Staubli VAL3: SettingGEN.dtx

num nCOLMAX = 39
num nCOLMIN
public num nColumn
public num nFocused
public num nListSize
num nROWMAX = 12
num nROWMIN
public num nRow
string sErrorMessage
string sErrorMsg[10]
  [1] = "An error has been detected in the Page library *\../*"
  [2] = "Variable sTxtBoxLen[*] has an illegal value"
  [3] = "Variable sTxtBoxPos[*] has an illegal value"
public string sFALSE = "FALSE"
public string sLabel[4]
  [0] = "-Calibrated pointer--"
  [1] = "-Event Logger --"
  [2] = "-Software --"
  [3] = "-Approach --"
public string sLabelPos[4]
  [0] = "0;0"
  [1] = "22;3"
  [2] = "22;0"
  [3] = "0;5"
public string sMenu = "; ; ; ENCODER DETECT CONVEYOR ; OK"
public string sTRUE = "TRUE"
public string sTitle
public string sTxtBoxAuthord[11]
  [0] = "0123456789.-"
  [1] = "0123456789.-"
  [2] = "0123456789.-"
  [3] = "0123456789.-"
  [4] = "0123456789.-"
  [5] = "0123456789.-"
  [6] = "0123456789.-"
  [7] = "0123456789.-"
  [8] = "0123456789.-"
  [9] = "0123456789"
  [10] = "0123456789"
public string sTxtBoxCaption[11]
  [0] = "X="
  [1] = "Y="
  [2] = "Z="
  [3] = "Rx="
  [4] = "Ry="
  [5] = "Rz="
  [6] = "X= "
  [7] = "Y= "
  [8] = "Z= "
  [9] = "Enable Log:"
  [10] = "Version:"
public string sTxtBoxLen[11]
  [0] = "7"
  [1] = "7"
  [2] = "7"
  [3] = "7"
  [4] = "7"
  [5] = "7"
  [6] = "4"
  [7] = "4"
  [8] = "4"
  [9] = "2"
  [10] = "9"
public string sTxtBoxPos[11]
  [0] = "0;1"
  [1] = "0;2"
  [2] = "0;3"
  [3] = "11;1"
  [4] = "11;2"
  [5] = "11;3"
  [6] = "0;6"
  [7] = "0;7"
  [8] = "0; 8"
  [9] = "22;4"
  [10] = "22;1"
public string sTxtBoxRange[11]
  [0] = "-1000;1000"
  [1] = "-1000;1000"
  [2] = "-1000;1000"
  [3] = "-180;180"
  [4] = "-180;180"
  [5] = "-180;180"
  [6] = "-100;100"
  [7] = "-100;100"
  [8] = "-100;100"
  [9] = "0;7"
  [10] = "0;0"
public string sTxtBoxType[11]
  [0] = "N"
  [1] = "N"
  [2] = "N"
  [3] = "N"
  [4] = "N"
  [5] = "N"
  [6] = "N"
  [7] = "N"
  [8] = "N"
  [9] = "N"
  [10] = "D"
public string sTxtBoxVal[11]
  [0] = "0"
  [1] = "0"
  [2] = "0"
  [3] = "0"
  [4] = "0"
  [5] = "0"
  [6] = "0"
  [7] = "0"
  [8] = "-100"
  [9] = "0"
  [10] = "0"
public string sListItem0
